TYPE U_Convert_UINT8 :
UNION
	nValue		:UINT;
	nBYTE		:BYTE;
END_UNION
END_TYPE

(* stored: Version 1.1.0.1, ProductVersion 3.1.4024.12
   DUT U_Convert_UINT8: Id {fc9aa775-5002-48e5-bdb1-66ac5602549d} *)
